// TIA Portal V20 export
// export: Created 2025-12-01T14:57:06.076993Z, ExportSetting None, DisplayName Totally Integrated Automation Portal, DisplayVersion V20 Update 3, DisplayName TIA Portal Openness, DisplayVersion V20 Update 3, DisplayName TIA Portal Version Control Interface, DisplayVersion V20 Update 3, DisplayName STEP 7 Professional, DisplayVersion V20 Update 3, DisplayName STEP 7 Safety, DisplayVersion V20 Update 2, DisplayName WinCC Basic/Comfort/Advanced, DisplayVersion V20 Update 3, DisplayName WinCC Professional, DisplayVersion V20 Update 3, DisplayName WinCC Unified, DisplayVersion V20 Update 3
FUNCTION "FC902_Decodifica_Selector" : Void   // FC902, LAD
TITLE = Digito de Selector
{ S7_Optimized_Access := 'FALSE' }
AUTHOR : GENERAL
NAME : 20150126
VERSION : 3.0
// stored: AutoNumber false, SetENOAutomatically false
   VAR_INPUT
      Bit_0 : Bool;
      Bit_1 : Bool;
      Bit_2 : Bool;
      Bit_3 : Bool;
   END_VAR
   VAR_OUTPUT
      Codigo : Word;
   END_VAR
BEGIN

REGION Network 1
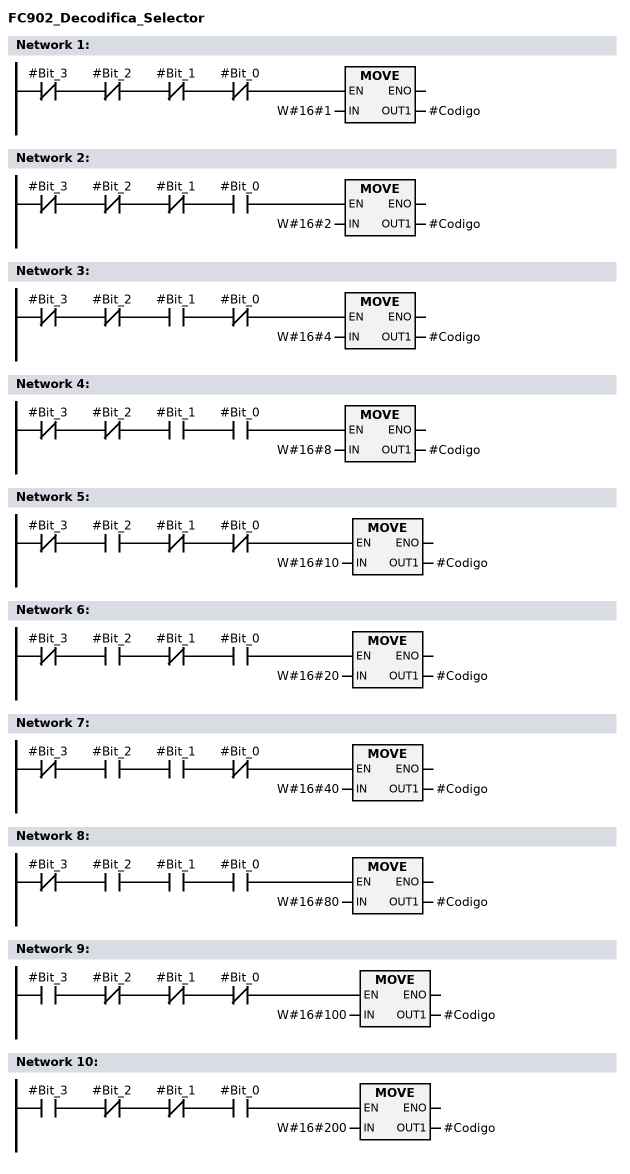
   RUNG wire#powerrail
      I_Contact( #Bit_3 )
      I_Contact( #Bit_2 )
      I_Contact( #Bit_1 )
      I_Contact( #Bit_0 )
      { S7_GenerateENO := "TRUE" } Move(in := W#16#1, out1 => #Codigo)
   END_RUNG
   // the same network as SCL:
   IF NOT #Bit_3 AND NOT #Bit_2 AND NOT #Bit_1 AND NOT #Bit_0 THEN #Codigo := W#16#1; END_IF;
END_REGION

REGION Network 2
   RUNG wire#powerrail
      I_Contact( #Bit_3 )
      I_Contact( #Bit_2 )
      I_Contact( #Bit_1 )
      Contact( #Bit_0 )
      { S7_GenerateENO := "TRUE" } Move(in := W#16#2, out1 => #Codigo)
   END_RUNG
   // the same network as SCL:
   IF NOT #Bit_3 AND NOT #Bit_2 AND NOT #Bit_1 AND #Bit_0 THEN #Codigo := W#16#2; END_IF;
END_REGION

REGION Network 3
   RUNG wire#powerrail
      I_Contact( #Bit_3 )
      I_Contact( #Bit_2 )
      Contact( #Bit_1 )
      I_Contact( #Bit_0 )
      { S7_GenerateENO := "TRUE" } Move(in := W#16#4, out1 => #Codigo)
   END_RUNG
   // the same network as SCL:
   IF NOT #Bit_3 AND NOT #Bit_2 AND #Bit_1 AND NOT #Bit_0 THEN #Codigo := W#16#4; END_IF;
END_REGION

REGION Network 4
   RUNG wire#powerrail
      I_Contact( #Bit_3 )
      I_Contact( #Bit_2 )
      Contact( #Bit_1 )
      Contact( #Bit_0 )
      { S7_GenerateENO := "TRUE" } Move(in := W#16#8, out1 => #Codigo)
   END_RUNG
   // the same network as SCL:
   IF NOT #Bit_3 AND NOT #Bit_2 AND #Bit_1 AND #Bit_0 THEN #Codigo := W#16#8; END_IF;
END_REGION

REGION Network 5
   RUNG wire#powerrail
      I_Contact( #Bit_3 )
      Contact( #Bit_2 )
      I_Contact( #Bit_1 )
      I_Contact( #Bit_0 )
      { S7_GenerateENO := "TRUE" } Move(in := W#16#10, out1 => #Codigo)
   END_RUNG
   // the same network as SCL:
   IF NOT #Bit_3 AND #Bit_2 AND NOT #Bit_1 AND NOT #Bit_0 THEN #Codigo := W#16#10; END_IF;
END_REGION

REGION Network 6
   RUNG wire#powerrail
      I_Contact( #Bit_3 )
      Contact( #Bit_2 )
      I_Contact( #Bit_1 )
      Contact( #Bit_0 )
      { S7_GenerateENO := "TRUE" } Move(in := W#16#20, out1 => #Codigo)
   END_RUNG
   // the same network as SCL:
   IF NOT #Bit_3 AND #Bit_2 AND NOT #Bit_1 AND #Bit_0 THEN #Codigo := W#16#20; END_IF;
END_REGION

REGION Network 7
   RUNG wire#powerrail
      I_Contact( #Bit_3 )
      Contact( #Bit_2 )
      Contact( #Bit_1 )
      I_Contact( #Bit_0 )
      { S7_GenerateENO := "TRUE" } Move(in := W#16#40, out1 => #Codigo)
   END_RUNG
   // the same network as SCL:
   IF NOT #Bit_3 AND #Bit_2 AND #Bit_1 AND NOT #Bit_0 THEN #Codigo := W#16#40; END_IF;
END_REGION

REGION Network 8
   RUNG wire#powerrail
      I_Contact( #Bit_3 )
      Contact( #Bit_2 )
      Contact( #Bit_1 )
      Contact( #Bit_0 )
      { S7_GenerateENO := "TRUE" } Move(in := W#16#80, out1 => #Codigo)
   END_RUNG
   // the same network as SCL:
   IF NOT #Bit_3 AND #Bit_2 AND #Bit_1 AND #Bit_0 THEN #Codigo := W#16#80; END_IF;
END_REGION

REGION Network 9
   RUNG wire#powerrail
      Contact( #Bit_3 )
      I_Contact( #Bit_2 )
      I_Contact( #Bit_1 )
      I_Contact( #Bit_0 )
      { S7_GenerateENO := "TRUE" } Move(in := W#16#100, out1 => #Codigo)
   END_RUNG
   // the same network as SCL:
   IF #Bit_3 AND NOT #Bit_2 AND NOT #Bit_1 AND NOT #Bit_0 THEN #Codigo := W#16#100; END_IF;
END_REGION

REGION Network 10
   RUNG wire#powerrail
      Contact( #Bit_3 )
      I_Contact( #Bit_2 )
      I_Contact( #Bit_1 )
      Contact( #Bit_0 )
      { S7_GenerateENO := "TRUE" } Move(in := W#16#200, out1 => #Codigo)
   END_RUNG
   // the same network as SCL:
   IF #Bit_3 AND NOT #Bit_2 AND NOT #Bit_1 AND #Bit_0 THEN #Codigo := W#16#200; END_IF;
END_REGION
END_FUNCTION
